// TIA Portal V20 export
DATA_BLOCK "DB_Msg"   // DB13
// stored: InstanceOfName FB_Msg, InstanceOfType FB
"FB_Msg"
   // VAR
   //    sSeverity : Byte;
   //    sMemoNumberOfActiveAlarms : DInt;
   //    sTON_On : TON_TIME;
   //    sTON_OFF { S7_SetPoint := 'True'} : TON_TIME;
   //    sPulseUpdateAlarms { S7_SetPoint := 'True'} : Bool;
   //    sRT_PulseUpdateAlarms : R_TRIG;
   // END_VAR
BEGIN
END_DATA_BLOCK
